(* CODESYS project PLC_Prj_RECOVERED_2025-07-21T23-08-57.project

Project tree, tasks and I/O mapping:
  Device : CODESYS Control Win V3 x64, CODESYS, version 3.5.21.10
    application Application
      libraries: Standard, 3.5.18.0 (System); CmpBitmapPool, * (System)
      task MainTask (cyclic, interval t#20ms, priority 1) calls POU_Main
      task VISU_TASK (cyclic, interval 100 ms, priority 31) calls VisuElems.Visu_Prg
      Symbols
      image pool ImagePool
      visualisation Visualization
      program POU_Main [LD]
  text list GlobalTextList
*)

// Device/Application/POU_Main
PROGRAM POU_Main
VAR
	Proximity: BOOL;
	BottleDetected: BOOL;
	ProximityTimer: TON;
	EjectBottle: BOOL;
	EjectRelay: BOOL;
	EjectionTimer: TON;
	exitScript: BOOL;
	SessionCounter: CTU;
	sessionNumber: INT;
	sessionNumber_pyProcess: INT;
	AcceptFlag: BOOL;
	EjectFlag: BOOL;
	HaveSolCmd : BOOL;
	HaveNewBottle : BOOL;
	R_Trig : R_Trig;
	AcceptFlag_TON : TON;
	EjectFlag_TON : TON;
	R_Trig_1 : R_Trig;
	R_Trig_2 : R_Trig;
END_VAR
VAR // added by the converter: edge detectors and wires of the graphical bodies
    _rt1 : R_TRIG;
    _w1, _w2 : BOOL;
END_VAR

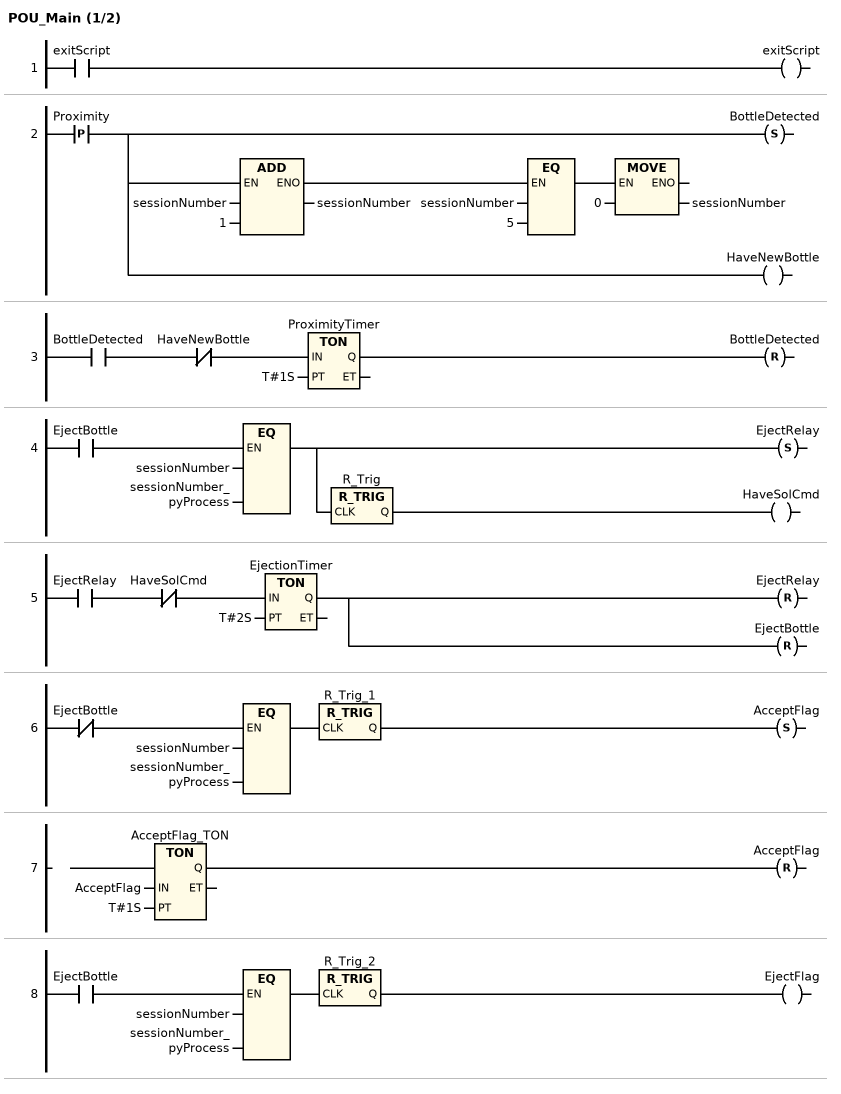
// NETWORK 1
exitScript := exitScript;

// NETWORK 2
_rt1(CLK := Proximity);
BottleDetected S= _rt1.Q;
_w1 := _rt1.Q;
IF _w1 THEN sessionNumber := sessionNumber + 1; END_IF
IF _w1 AND sessionNumber = 5 THEN sessionNumber := 0; END_IF
HaveNewBottle := _rt1.Q;

// NETWORK 3
ProximityTimer(IN := BottleDetected AND NOT HaveNewBottle, PT := T#1S); // TON
BottleDetected R= ProximityTimer.Q;

// NETWORK 4
_w2 := EjectBottle AND sessionNumber = sessionNumber_pyProcess;
EjectRelay S= _w2;
R_Trig(CLK := _w2);
HaveSolCmd := R_Trig.Q;

// NETWORK 5
EjectionTimer(IN := EjectRelay AND NOT HaveSolCmd, PT := T#2S); // TON
EjectRelay R= EjectionTimer.Q;
EjectBottle R= EjectionTimer.Q;

// NETWORK 6
R_Trig_1(CLK := NOT EjectBottle AND sessionNumber = sessionNumber_pyProcess); // R_TRIG
AcceptFlag S= R_Trig_1.Q;

// NETWORK 7
AcceptFlag_TON(IN := AcceptFlag, PT := T#1S); // TON
AcceptFlag R= AcceptFlag_TON.Q;

// NETWORK 8
R_Trig_2(CLK := EjectBottle AND sessionNumber = sessionNumber_pyProcess); // R_TRIG
EjectFlag := R_Trig_2.Q;

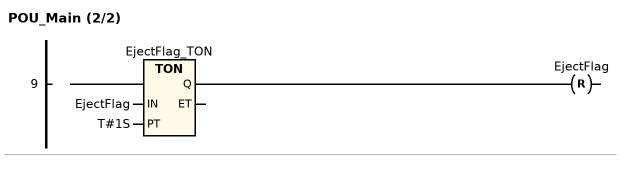
// NETWORK 9
EjectFlag_TON(IN := EjectFlag, PT := T#1S); // TON
EjectFlag R= EjectFlag_TON.Q;

END_PROGRAM

// Device/Application/Visualization
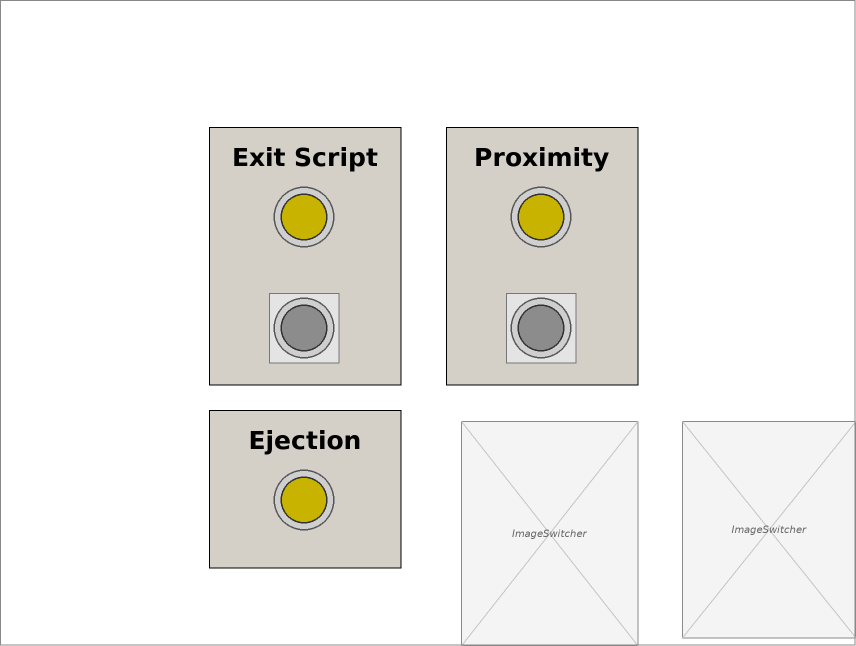
VISUALIZATION Visualization  // 856x646
    RoundedRectangle (209,127 192x258)
    PushSwitch (269,293 70x70), variable: POU_Main.exitScript, behaviour: TAP, style: Switch-PushSwitch-Gray
    Lamp1 (269,182 70x70), variable: POU_Main.exitScript, style: Lamp-Lamp1-Yellow
    Label (209,142 192x30), "Exit Script"
    RoundedRectangle (446,127 192x258)
    PushSwitch (506,293 70x70), variable: POU_Main.Proximity, behaviour: TAP, style: Switch-PushSwitch-Gray
    Lamp1 (506,182 70x70), variable: POU_Main.BottleDetected, style: Lamp-Lamp1-Yellow
    Label (446,142 192x30), "Proximity"
    RoundedRectangle (209,410 192x158)
    Lamp1 (269,465 70x70), variable: POU_Main.EjectRelay, style: Lamp-Lamp1-Yellow
    Label (209,425 192x30), "Ejection"
    ImageSwitcher (461,421 177x225), variable: POU_Main.AcceptFlag, background image: ImagePool.2, behaviour: TOGGLE
    ImageSwitcher (682,421 174x217), variable: POU_Main.EjectFlag, background image: ImagePool.1, behaviour: TOGGLE
END_VISUALIZATION
